SUBAPPLICATION mapping_NumericValue (* Subapplication Type *)
  (* Standard: 61499-2 *)
  (* Version 1.0, 2023-01-29, Franz *)
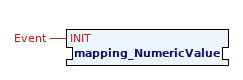
  EVENT_INPUT
    INIT;
  END_EVENT
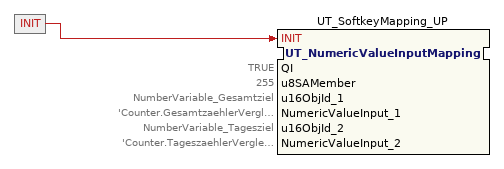
  FBS
    UT_SoftkeyMapping_UP : UT_NumericValueInputMapping(QI := TRUE, u8SAMember := 255, u16ObjId_1 := NumberVariable_Gesamtziel, NumericValueInput_1 := 'Counter.GesamtzaehlerVergleich.IN_NumberVariable_Gesamtziel', u16ObjId_2 := NumberVariable_Tagesziel, NumericValueInput_2 := 'Counter.TageszaehlerVergleich.IN_NumberVariable_Tagesziel');
  END_FBS
  EVENT_CONNECTIONS
    INIT TO UT_SoftkeyMapping_UP.INIT;
  END_CONNECTIONS
END_SUBAPPLICATION
